Universal Robots PolyScope program: trigger_reduced_mode_feature_214.urp

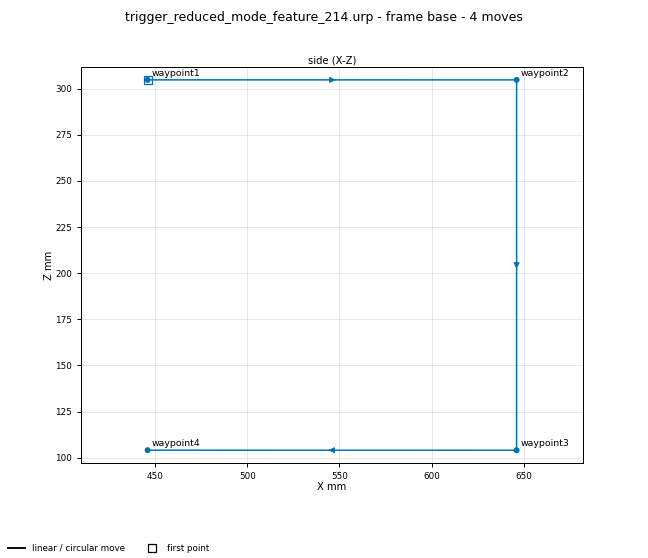
[picture p0: tool path of trigger_reduced_mode_feature_214.urp in frame base, 4 of 4 moves have a stored position in this frame; points joined in program order, loops and branches not executed]
Program trigger_reduced_mode_feature_214 (createdIn=3.2.19293 lastSavedIn=3.2.19293 directory=/programs installation=default robotSerialNumber=2015351391)
Calibrated DH parameters: a=[0.000352, -0.161198, -0.373486, 0.00005, 0.000049, 0]; d=[0.089268, 352.477598, -320.08558, -32.281492, 0.094939, 0.082518]; alpha=[1.570728, 0.001116, -0.003686, 1.571189, -1.570572, 0]; deltaTheta=[-0.000012, 1.181849, -1.491165, 0.309495, -0.000007, 0.000025]
Robot Program (runOnlyOnce=false motionType=MoveJ speed=1.047198 acceleration=1.396263 recalculateMotions=false)
  MoveL speed 1500 mm/s, acceleration 2500 mm/s^2 (recalculateMotions=false) feature=Base
    Waypoint waypoint1: TCP in base x=445.967 y=-138.792 z=304.781 mm, rx=0.6753 ry=1.4825 rz=0.4858 rad; joints [-1.05, -87.533, -141.535, 46.939, 84.789, 132.588] deg; flange x=321.882 y=-124.718 z=309.335 mm, rx=0.6755 ry=1.4826 rz=0.4858 rad
    Waypoint waypoint2: TCP in base x=646.015 y=-138.806 z=304.767 mm, rx=0.6754 ry=1.4824 rz=0.4858 rad; joints [-0.546, -110.941, -112.285, 41.104, 84.295, 132.599] deg; flange x=521.882 y=-124.733 z=309.338 mm, rx=0.6755 ry=1.4825 rz=0.4857 rad
    Waypoint waypoint3: TCP in base x=646 y=-138.859 z=103.996 mm, rx=0.6755 ry=1.4825 rz=0.4856 rad; joints [-0.573, -135.798, -114.374, 68.037, 84.363, 132.711] deg; flange x=521.883 y=-124.748 z=108.584 mm, rx=0.6755 ry=1.4825 rz=0.4856 rad
    Waypoint waypoint4: TCP in base x=445.994 y=-138.876 z=104.026 mm, rx=0.6755 ry=1.4823 rz=0.4857 rad; joints [-1.141, -131.796, -144.721, 94.378, 84.918, 132.781] deg; flange x=321.882 y=-124.765 z=108.58 mm, rx=0.6754 ry=1.4825 rz=0.4857 rad
